// TIA Portal V20 export
TYPE "DigitalInput_DT"
   STRUCT
      SWStatus : Bool;   // Software status use in PLC code
      SWPositiveFront : Bool;   // Positive front of software status
      SWNegativeFront : Bool;   // Negative front of sofware status
      HWStatus : Bool;   // Hardware status directly from physical input
   END_STRUCT;
END_TYPE
